Fanuc KAREL source: ko00108.KL

PROGRAM KO00108
%STACKSIZE=65535
%PRIORITY=65535
%NOLOCKGROUP
VAR
A : REAL
B : REAL
OUT : REAL
BEGIN
A=1
B=2
-- UNRESOLVED_PC line 10 opcodes [27 22 22 76 23] marker_code=30
END KO00108
